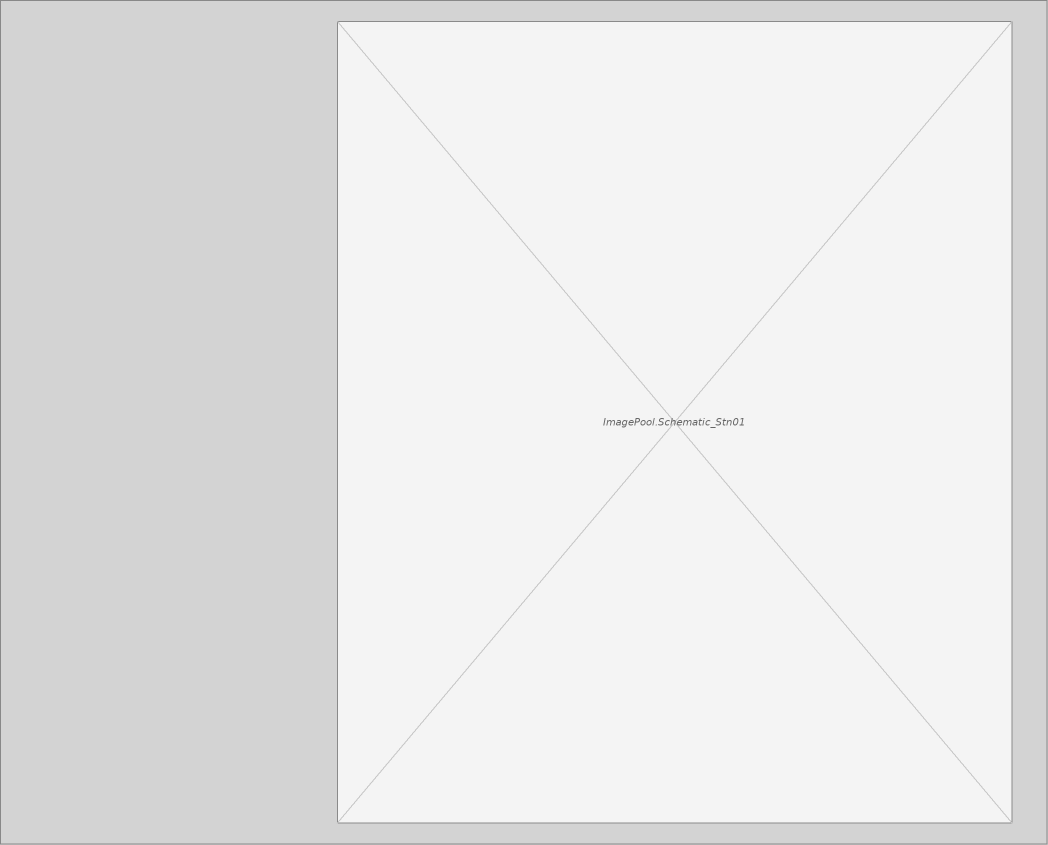
VISUALIZATION Recipe_Station12  // 1048x845
    Rectangle (0,0 1048x845)
    Image (337,21 675x802), image: ImagePool.Schematic_Stn01
END_VISUALIZATION

(* stored: Version 1.1.0.1, ProductVersion 3.1.4024.12
   Visu Recipe_Station12: Id {f2149da8-0984-433c-a9c1-c8c3456d94c7} *)
